FUNCTION_BLOCK FB_Bloque
VAR_INPUT
	Tcheck: TIME := T#1S;
	Treset: TIME := T#1S;
END_VAR
VAR_OUTPUT
END_VAR
VAR
	pulsador AT %I*: BOOL; 
	verificador_abajo AT %I*: BOOL;
	motor AT %Q*: BOOL;
	lampara AT %Q*: BOOL;
	pieza_ok AT %Q*: BOOL;
END_VAR

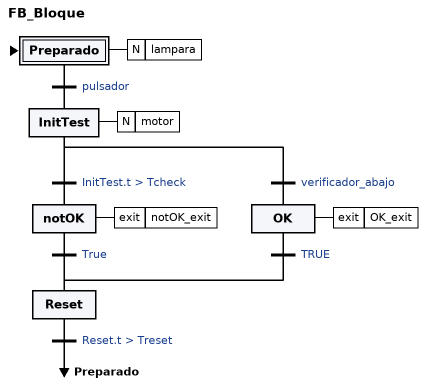
INITIAL_STEP Preparado:
    lampara(N);
END_STEP
TRANSITION FROM Preparado TO InitTest
    := pulsador;
END_TRANSITION
STEP InitTest:
    motor(N);
END_STEP
TRANSITION FROM InitTest TO notOK
    := InitTest.t > Tcheck;
END_TRANSITION
STEP notOK:
    notOK_exit(P0);  // exit action
END_STEP
TRANSITION FROM notOK TO Reset
    := True;
END_TRANSITION
TRANSITION FROM InitTest TO OK
    := verificador_abajo;
END_TRANSITION
STEP OK:
    OK_exit(P0);  // exit action
END_STEP
TRANSITION FROM OK TO Reset
    := TRUE;
END_TRANSITION
STEP Reset:
END_STEP
TRANSITION FROM Reset TO Preparado
    := Reset.t > Treset;
END_TRANSITION

ACTION notOK_exit:
pieza_ok := FALSE;
END_ACTION

ACTION OK_exit:
pieza_ok := false;
END_ACTION

END_FUNCTION_BLOCK

(* stored: Version 1.1.0.1, ProductVersion 3.1.4024.12
   POU FB_Bloque: Id {0c102bf0-d2ee-4790-8611-bbcb80572984}, SpecialFunc None
   Action notOK_exit: Id {7c7983fe-474f-4382-8939-3f4e8ea06912}
   Action OK_exit: Id {6923b980-9502-4e1c-97e4-e82bb8b6c6b3} *)
